// TIA Portal V16 export
// export: Created 2024-09-05T17:39:19.835415Z, ExportSetting WithDefaults, DisplayName Totally Integrated Automation Portal, DisplayVersion V16 Update 6, DisplayName TIA Portal Version Control Interface, DisplayVersion V16 Update 2, DisplayName TIA Portal Openness, DisplayVersion V16 Update 6, DisplayName STEP 7 Professional, DisplayVersion V16 Update 6, DisplayName STEP 7 Safety, DisplayVersion V16, DisplayName WinCC Advanced, DisplayVersion V16 Update 6
FUNCTION_BLOCK "sq_carousel_st1"   // FB39, GRAPH
VERSION : 0.1
// stored: AcknowledgeErrorsRequired true, AutoNumber true, GraphVersion 6.0, InitialValuesAcquisition false, IsIECCheckEnabled false, LanguageInNetworks LAD, LockOperatingMode false, PermanentILProcessingInMANMode false, SetENOAutomatically false, SkipSteps false, UDAEnableTagReadback false, WithAlarmHandling true
   // inherited from GRAPH_BASE
   VAR
      OFF_SQ_BASE : Bool;
   END_VAR
   VAR_INPUT
      OFF_SQ { ExternalAccessible := 'False'; ExternalVisible := 'False'; ExternalWritable := 'False'} : Bool := false;   // Turn sequence off
      INIT_SQ { ExternalAccessible := 'False'; ExternalVisible := 'False'; ExternalWritable := 'False'} : Bool := false;   // Set sequence to initial state
      ACK_EF { ExternalAccessible := 'False'; ExternalVisible := 'False'; ExternalWritable := 'False'} : Bool := false;   // Acknowledge all errors and faults
      S_PREV { ExternalAccessible := 'False'; ExternalVisible := 'False'; ExternalWritable := 'False'} : Bool := false;   // Output previous step in parameter S_NO
      S_NEXT { ExternalAccessible := 'False'; ExternalVisible := 'False'; ExternalWritable := 'False'} : Bool := false;   // Indicate next step in parameter S_NO
      SW_AUTO { ExternalAccessible := 'False'; ExternalVisible := 'False'; ExternalWritable := 'False'} : Bool := false;   // Automatic mode
      SW_TAP { ExternalAccessible := 'False'; ExternalVisible := 'False'; ExternalWritable := 'False'} : Bool := false;   // Semiautomatic/switch with transition
      SW_TOP { ExternalAccessible := 'False'; ExternalVisible := 'False'; ExternalWritable := 'False'} : Bool := false;   // Semiautomatic/ignore transition
      SW_MAN { ExternalAccessible := 'False'; ExternalVisible := 'False'; ExternalWritable := 'False'} : Bool := false;   // Manual mode
      S_SEL { ExternalAccessible := 'False'; ExternalVisible := 'False'; ExternalWritable := 'False'} : Int := 0;   // Select step to be output to S_NO
      S_ON { ExternalAccessible := 'False'; ExternalVisible := 'False'; ExternalWritable := 'False'} : Bool := false;   // Activate step indicated in S_NO
      S_OFF { ExternalAccessible := 'False'; ExternalVisible := 'False'; ExternalWritable := 'False'} : Bool := false;   // Deactivate step indicated S_NO
      T_PUSH { ExternalAccessible := 'False'; ExternalVisible := 'False'; ExternalWritable := 'False'} : Bool := false;   // Enable transition to switch in semi automatic mode
   END_VAR
   VAR_OUTPUT
      S_NO { ExternalAccessible := 'False'; ExternalVisible := 'False'; ExternalWritable := 'False'} : Int := 0;   // Step number
      S_MORE { ExternalAccessible := 'False'; ExternalVisible := 'False'; ExternalWritable := 'False'} : Bool := false;   // More steps are available and can be shown in S_NO
      S_ACTIVE { ExternalAccessible := 'False'; ExternalVisible := 'False'; ExternalWritable := 'False'} : Bool := false;   // Step indicated in S_NO is active
      ERR_FLT { ExternalAccessible := 'False'; ExternalVisible := 'False'; ExternalWritable := 'False'} : Bool := false;   // Interlock or supervision group error
      AUTO_ON { ExternalAccessible := 'False'; ExternalVisible := 'False'; ExternalWritable := 'False'} : Bool := false;   // Automatic mode is active
      TAP_ON { ExternalAccessible := 'False'; ExternalVisible := 'False'; ExternalWritable := 'False'} : Bool := false;   // Semiautomatic mode/step with transition enabled
      TOP_ON { ExternalAccessible := 'False'; ExternalVisible := 'False'; ExternalWritable := 'False'} : Bool := false;   // Semiautomatic mode/ignore transition enabled
      MAN_ON { ExternalAccessible := 'False'; ExternalVisible := 'False'; ExternalWritable := 'False'} : Bool := false;   // Manual mode is active
   END_VAR
   VAR
      dummy : Bool;
      start : Bool;
      base : Bool;
      startEmpty : Bool;
   END_VAR
   VAR_TEMP   // added for the SCL form of the ladder/FBD networks
      _w1 : Bool;
      _w2 : Bool;
   END_VAR
BEGIN
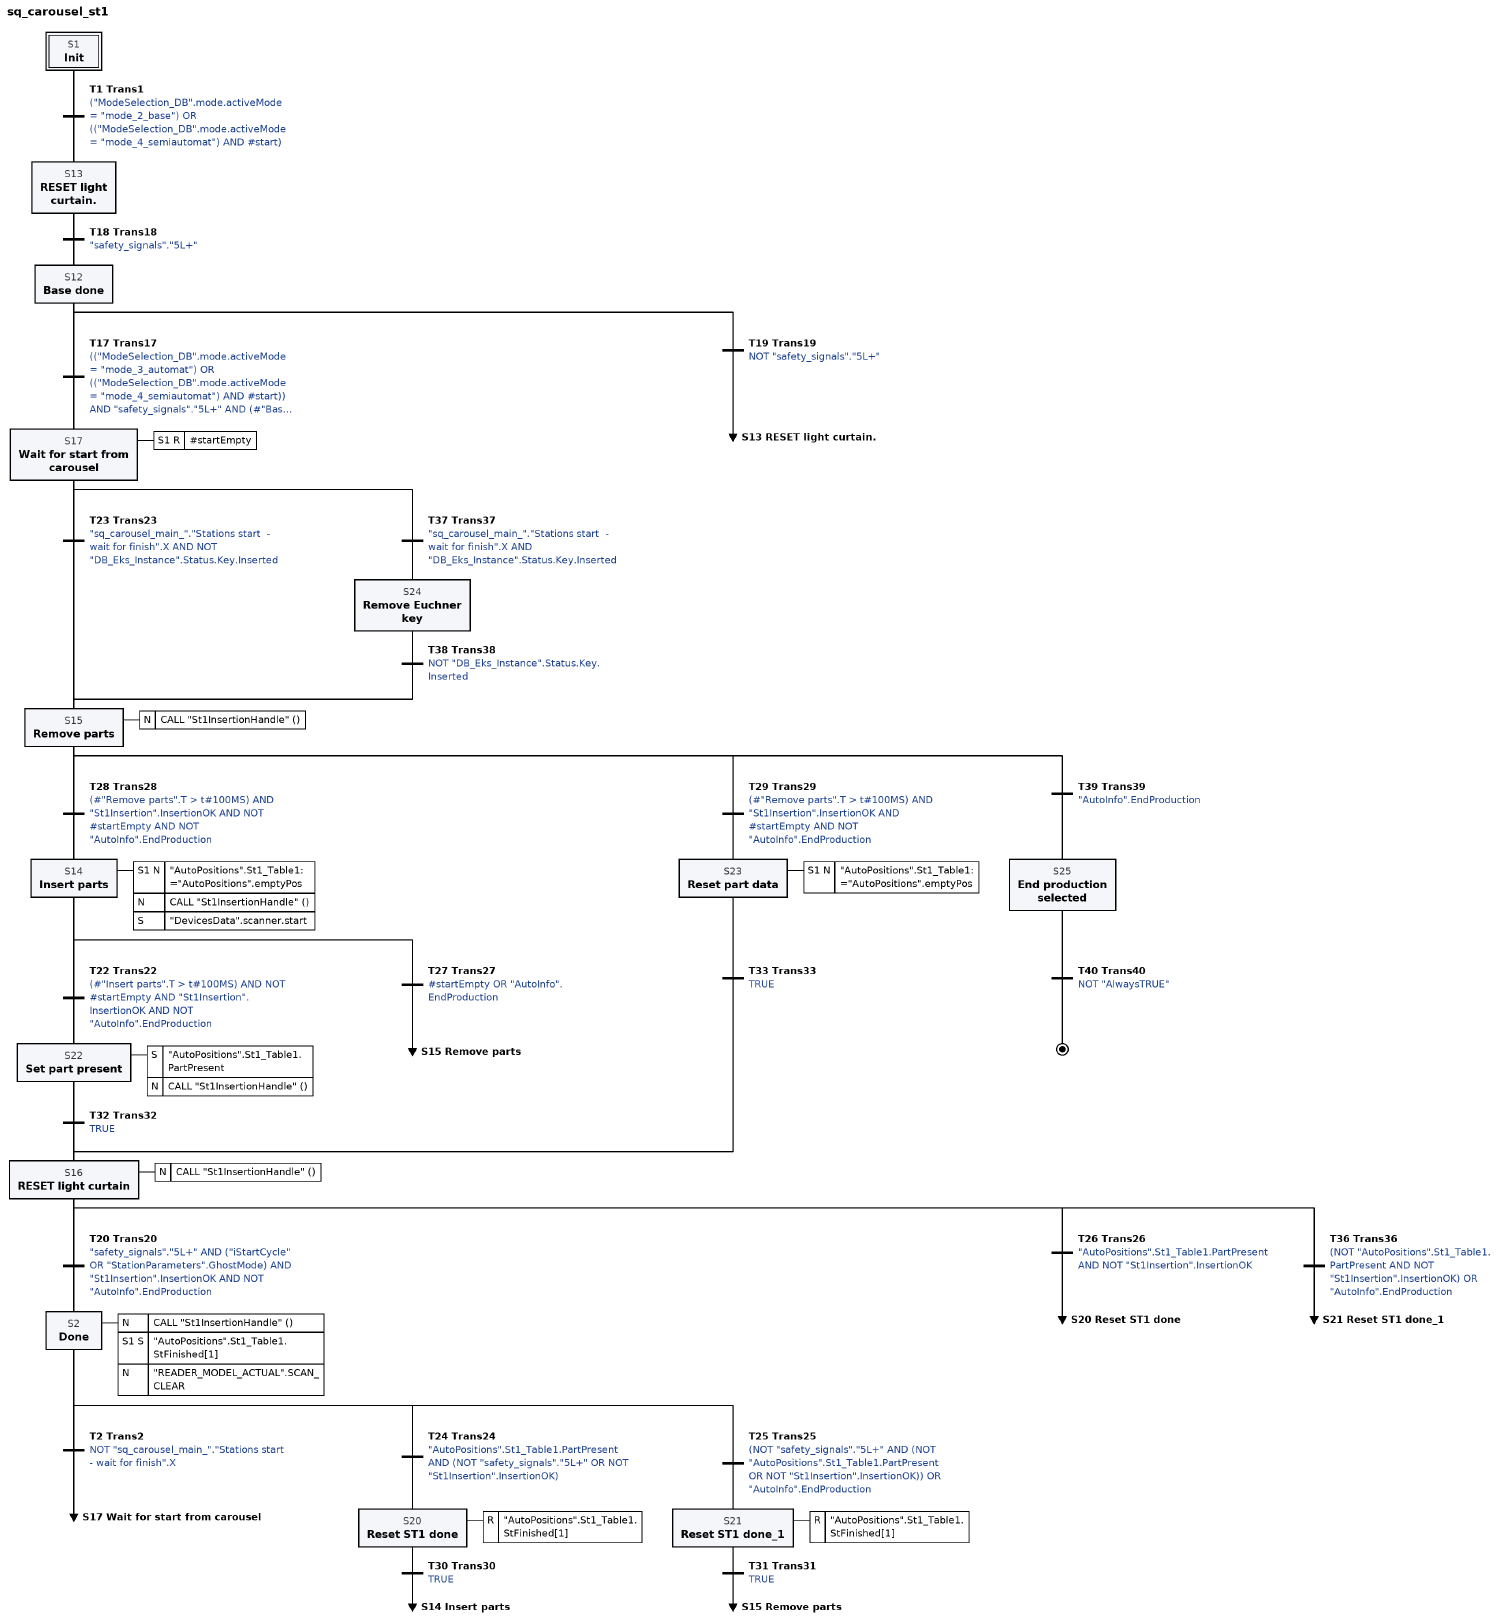
   // permanent pre-instructions
   NETWORK 1
      #base := TRUE;
   NETWORK 2
      "St1Insertion".ExpectedSensors := "St1Insertion".EmptyBits;
      #_w1 := ("ModeSelection_DB".mode.activeMode = "mode_3_automat") OR ("ModeSelection_DB".mode.activeMode = "mode_4_semiautomat");
      IF #_w1 THEN "St1Insertion".UsedSensors := "St1Insertion".FullBits; END_IF;
      IF NOT #_w1 THEN "St1Insertion".UsedSensors := "St1Insertion".EmptyBits; END_IF;
      #_w2 := ("AutoPositions".St1_Table1.PartPresent OR #"Insert parts".X) AND NOT #startEmpty AND NOT "StationParameters".GhostMode AND NOT #"Remove parts".X;
      IF #_w2 THEN
          MOVE_BLK(IN := "DB_ProductionProgramActual".Program.St1Insertion[1],
                   COUNT := 20,
                   OUT => "St1Insertion".ExpectedSensors[1]);
          MOVE_BLK(IN := "DB_ProductionProgramActual".Program.St1InsertionUsed[1],
                   COUNT := 20,
                   OUT => "St1Insertion".UsedSensors[1]);
      END_IF;
      "St1InsertionHandle"();

   // sequencer 1
   INITIAL_STEP Init:   // S1, max time T#10S, warning time T#7S
   END_STEP
   TRANSITION Trans1 FROM Init TO "RESET light curtain."   // T1
      := ("ModeSelection_DB".mode.activeMode = "mode_2_base") OR (("ModeSelection_DB".mode.activeMode = "mode_4_semiautomat") AND #start);
   END_TRANSITION
   STEP Done:   // S2, max time T#10S, warning time T#7S
              N    CALL "St1InsertionHandle" ()
          S1  S    "AutoPositions".St1_Table1.StFinished[1]
              N    "READER_MODEL_ACTUAL".SCAN_CLEAR
   END_STEP
   TRANSITION Trans2 FROM Done TO "Wait for start from carousel"   // T2, jump
      := NOT "sq_carousel_main_"."Stations start  - wait for finish".X;
   END_TRANSITION
   TRANSITION Trans24 FROM Done TO "Reset ST1 done"   // T24
      := "AutoPositions".St1_Table1.PartPresent AND (NOT "safety_signals"."5L+" OR NOT "St1Insertion".InsertionOK);
   END_TRANSITION
   TRANSITION Trans25 FROM Done TO "Reset ST1 done_1"   // T25
      := (NOT "safety_signals"."5L+" AND (NOT "AutoPositions".St1_Table1.PartPresent OR NOT "St1Insertion".InsertionOK)) OR "AutoInfo".EndProduction;
   END_TRANSITION
   STEP "Base done":   // S12, max time T#10S, warning time T#7S
   END_STEP
   TRANSITION Trans17 FROM "Base done" TO "Wait for start from carousel"   // T17
      := (("ModeSelection_DB".mode.activeMode = "mode_3_automat") OR (("ModeSelection_DB".mode.activeMode = "mode_4_semiautomat") AND #start)) AND "safety_signals"."5L+" AND (#"Base done".T > t#2000MS);
   END_TRANSITION
   TRANSITION Trans19 FROM "Base done" TO "RESET light curtain."   // T19, jump
      := NOT "safety_signals"."5L+";
   END_TRANSITION
   STEP "RESET light curtain.":   // S13, max time T#10S, warning time T#7S
   END_STEP
   TRANSITION Trans18 FROM "RESET light curtain." TO "Base done"   // T18
      := "safety_signals"."5L+";
   END_TRANSITION
   STEP "Insert parts":   // S14, max time T#10S, warning time T#7S
          S1  N    "AutoPositions".St1_Table1:="AutoPositions".emptyPos
              N    CALL "St1InsertionHandle" ()
              S    "DevicesData".scanner.start
   END_STEP
   TRANSITION Trans22 FROM "Insert parts" TO "Set part present"   // T22
      := (#"Insert parts".T > t#100MS) AND NOT #startEmpty AND "St1Insertion".InsertionOK AND NOT "AutoInfo".EndProduction;
   END_TRANSITION
   TRANSITION Trans27 FROM "Insert parts" TO "Remove parts"   // T27, jump
      := #startEmpty OR "AutoInfo".EndProduction;
   END_TRANSITION
   STEP "Remove parts":   // S15, max time T#10S, warning time T#7S
              N    CALL "St1InsertionHandle" ()
   END_STEP
   TRANSITION Trans28 FROM "Remove parts" TO "Insert parts"   // T28
      := (#"Remove parts".T > t#100MS) AND "St1Insertion".InsertionOK AND NOT #startEmpty AND NOT "AutoInfo".EndProduction;
   END_TRANSITION
   TRANSITION Trans29 FROM "Remove parts" TO "Reset part data"   // T29
      := (#"Remove parts".T > t#100MS) AND "St1Insertion".InsertionOK AND #startEmpty AND NOT "AutoInfo".EndProduction;
   END_TRANSITION
   TRANSITION Trans39 FROM "Remove parts" TO "End production selected"   // T39
      := "AutoInfo".EndProduction;
   END_TRANSITION
   STEP "RESET light curtain":   // S16, max time T#10S, warning time T#7S
              N    CALL "St1InsertionHandle" ()
   END_STEP
   TRANSITION Trans20 FROM "RESET light curtain" TO Done   // T20
      := "safety_signals"."5L+" AND ("iStartCycle" OR "StationParameters".GhostMode) AND "St1Insertion".InsertionOK AND NOT "AutoInfo".EndProduction;
   END_TRANSITION
   TRANSITION Trans26 FROM "RESET light curtain" TO "Reset ST1 done"   // T26, jump
      := "AutoPositions".St1_Table1.PartPresent AND NOT "St1Insertion".InsertionOK;
   END_TRANSITION
   TRANSITION Trans36 FROM "RESET light curtain" TO "Reset ST1 done_1"   // T36, jump
      := (NOT "AutoPositions".St1_Table1.PartPresent AND NOT "St1Insertion".InsertionOK) OR "AutoInfo".EndProduction;
   END_TRANSITION
   STEP "Wait for start from carousel":   // S17, max time T#10S, warning time T#7S
          S1  R    #startEmpty
   END_STEP
   TRANSITION Trans23 FROM "Wait for start from carousel" TO "Remove parts"   // T23
      := "sq_carousel_main_"."Stations start  - wait for finish".X AND NOT "DB_Eks_Instance".Status.Key.Inserted;
   END_TRANSITION
   TRANSITION Trans37 FROM "Wait for start from carousel" TO "Remove Euchner key"   // T37
      := "sq_carousel_main_"."Stations start  - wait for finish".X AND "DB_Eks_Instance".Status.Key.Inserted;
   END_TRANSITION
   STEP "Reset ST1 done":   // S20, max time T#10S, warning time T#7S
              R    "AutoPositions".St1_Table1.StFinished[1]
   END_STEP
   TRANSITION Trans30 FROM "Reset ST1 done" TO "Insert parts"   // T30, jump
      := TRUE;
   END_TRANSITION
   STEP "Reset ST1 done_1":   // S21, max time T#10S, warning time T#7S
              R    "AutoPositions".St1_Table1.StFinished[1]
   END_STEP
   TRANSITION Trans31 FROM "Reset ST1 done_1" TO "Remove parts"   // T31, jump
      := TRUE;
   END_TRANSITION
   STEP "Set part present":   // S22, max time T#10S, warning time T#7S
              S    "AutoPositions".St1_Table1.PartPresent
              N    CALL "St1InsertionHandle" ()
   END_STEP
   TRANSITION Trans32 FROM "Set part present" TO "RESET light curtain"   // T32
      := TRUE;
   END_TRANSITION
   STEP "Reset part data":   // S23, max time T#10S, warning time T#7S
          S1  N    "AutoPositions".St1_Table1:="AutoPositions".emptyPos
   END_STEP
   TRANSITION Trans33 FROM "Reset part data" TO "RESET light curtain"   // T33
      := TRUE;
   END_TRANSITION
   STEP "Remove Euchner key":   // S24, max time T#10S, warning time T#7S
   END_STEP
   TRANSITION Trans38 FROM "Remove Euchner key" TO "Remove parts"   // T38
      := NOT "DB_Eks_Instance".Status.Key.Inserted;
   END_TRANSITION
   STEP "End production selected":   // S25, max time T#10S, warning time T#7S
   END_STEP
   TRANSITION Trans40 FROM "End production selected" TO END   // T40
      := NOT "AlwaysTRUE";
   END_TRANSITION
END_FUNCTION_BLOCK
